// TwinCAT 3 PLC project PLCSim
// ProgramVersion: 3.1.4026.21
// libraries:
//   Tc2_Standard, * (Beckhoff Automation GmbH)
//   Tc2_System, * (Beckhoff Automation GmbH)
//   Tc3_Module, * (Beckhoff Automation GmbH)
//   VisuSymbols,newest,System
// project tree:
//   / GlobalTextList.TcGTLO, PlcTask.TcTTO, Visualization Manager.TcVMO (not stored)
//   GVLs/ GVL.TcGVL (not stored)
//   POUs/ AGV.TcPOU (not stored), MAIN.TcPOU, Process.TcPOU
//   VISUs/ AGVSimulator.TcVIS
// real-time tasks:
//   TASK PlcTask: cycle T#20ms, priority 20, ADS port 350
// variable links:
//   PLCSim/PLCSim Instance <-> PLCStudent/PLCStudent Instance
//     PlcTask Inputs/GVL.iiGotoPos <-> PlcTask Outputs/GVL.iiGotoPos
//     PlcTask Inputs/GVL.ixPLCStrobe <-> PlcTask Outputs/GVL.ixPLCStrobe
//     PlcTask Outputs/GVL.qiAtPos <-> PlcTask Inputs/GVL.iiAtPos
//     PlcTask Outputs/GVL.qxAGVStrobe <-> PlcTask Inputs/GVL.ixAGVStrobe

CONFIGURATION PLCSim
    RESOURCE PLC ON TwinCAT3
        TASK PlcTask(INTERVAL := T#20ms, PRIORITY := 20);
        PROGRAM MAIN WITH PlcTask : MAIN;
    END_RESOURCE
END_CONFIGURATION

// ---- POUs/MAIN.TcPOU
PROGRAM MAIN

VAR

END_VAR

Process();

END_PROGRAM

// ---- POUs/Process.TcPOU
PROGRAM Process
VAR
	fbAGV : AGV;
END_VAR

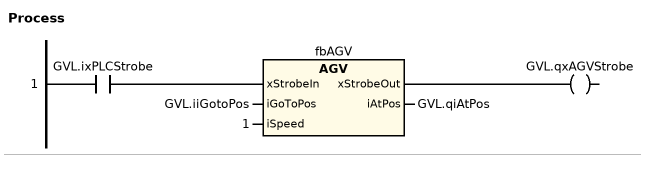
// NETWORK 1
fbAGV(xStrobeIn := GVL.ixPLCStrobe, iGoToPos := GVL.iiGotoPos, iSpeed := 1, iAtPos => GVL.qiAtPos); // AGV
GVL.qxAGVStrobe := fbAGV.xStrobeOut;

END_PROGRAM

// ---- GlobalTextList.TcGTLO
TEXTLIST GlobalTextList
  546 = 'AGV'
  738 = 'ERROR'
  838 = 'HOME'
  505 = 'Pos A'
  284 = 'Pos AD'
  908 = 'Pos B'
  412 = 'Pos C'
  547 = 'Pos D'
  315 = 'University West'
  428 = 'Ver 2.0'
END_TEXTLIST

// ---- VISUs/AGVSimulator.TcVIS
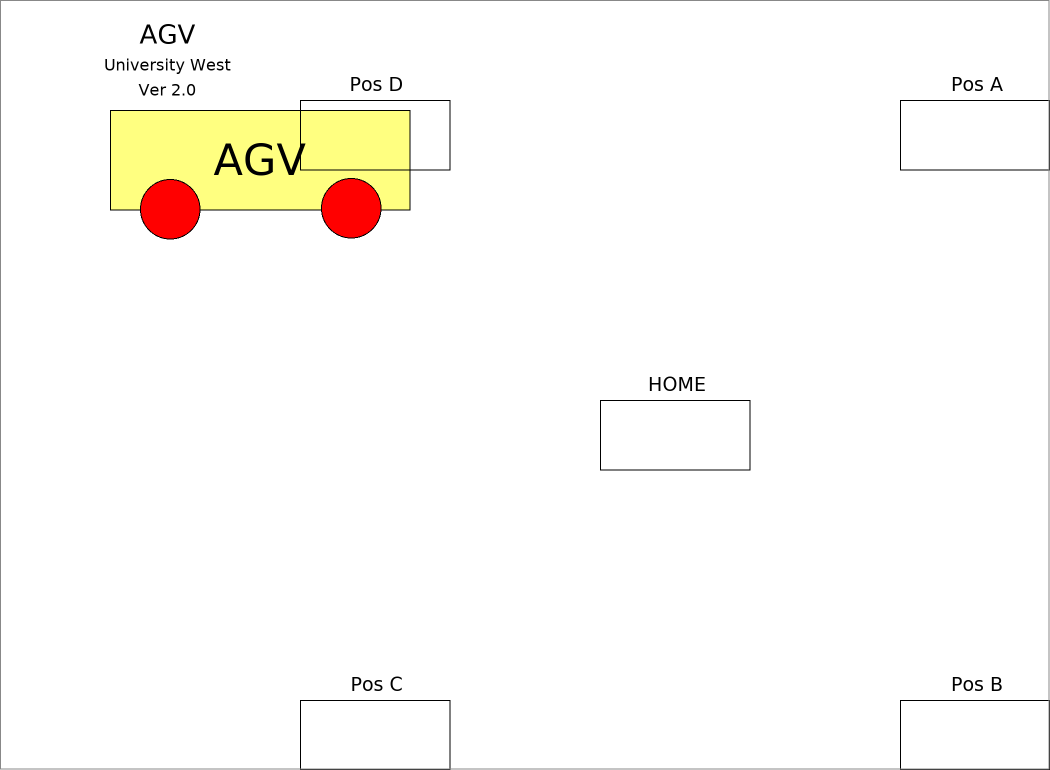
VISUALIZATION AGVSimulator  // 1050x770
    Group (110,110 130x50)
        p3560616238: Process.fbAGV.iAtPos_X
        p2738717112: Process.fbAGV.iAtPos_Y
        RoundedRectangle (0,0 300x100), "AGV"
        Ellipse (30,69 60x60)
        Ellipse (211,68 60x60)
    RoundedRectangle (300,100 150x70)
    RoundedRectangle (900,100 150x70)
    RoundedRectangle (600,400 150x70)
    RoundedRectangle (900,700 150x70)
    RoundedRectangle (300,700 150x70)
    Rectangle (330,670 94x29), "Pos C"
    Rectangle (930,670 94x29), "Pos B"
    Rectangle (930,70 94x29), "Pos A"
    Rectangle (330,70 93x29), "Pos D"
    Rectangle (630,370 94x29), "HOME"
    Rectangle (130,370 94x29), "ERROR", invisible if: NOT Process.fbAGV.xError
    Rectangle (80,20 175x29), "AGV"
    Rectangle (80,50 175x30), "University West"
    Rectangle (80,75 175x30), "Ver 2.0"
    RoundedRectangle (107,356 144x54), invisible if: Process.fbAGV.xError
END_VISUALIZATION
